FUNCTION POU : INT
VAR_INPUT
END_VAR
VAR
END_VAR

// NETWORK 1

// NETWORK 2

// NETWORK 3

END_FUNCTION

(* stored: Version 1.1.0.1, ProductVersion 3.1.4018.2
   POU POU: Id {c68534b8-4ccb-4393-a9ee-a4b4d0184c9c}, SpecialFunc None *)
